(* PLC project Unnamed, Unknown Unnamed 1 *)
(* stored: creationDateTime 2019-08-06T14:23:42, modificationDateTime 2023-08-18T11:29:36 *)

PROGRAM MainStuff
  VAR
    var0 : HMI_REAL;
    var1 : HMI_SINT;
    var2 : HMI_INT;
    var3 : HMI_DINT;
    var4 : HMI_LINT;
    var5 : HMI_USINT;
    var6 : HMI_UINT;
    var7 : HMI_UDINT;
    var8 : HMI_ULINT;
    var9 : HMI_UDINT;
  END_VAR

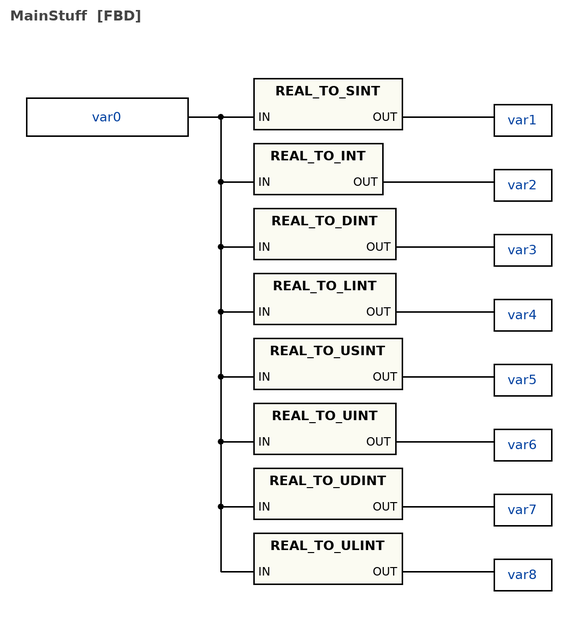
(* FBD diagram, written out as Structured Text *)
var1 := REAL_TO_SINT(var0);
var2 := REAL_TO_INT(var0);
var3 := REAL_TO_DINT(var0);
var4 := REAL_TO_LINT(var0);
var5 := REAL_TO_USINT(var0);
var6 := REAL_TO_UINT(var0);
var7 := REAL_TO_UDINT(var0);
var8 := REAL_TO_ULINT(var0);
END_PROGRAM

CONFIGURATION config
  RESOURCE resource1 ON PLC
    TASK task0(INTERVAL := T#20ms, PRIORITY := 0);
    PROGRAM instance0 WITH task0 : MainStuff;
  END_RESOURCE
END_CONFIGURATION
